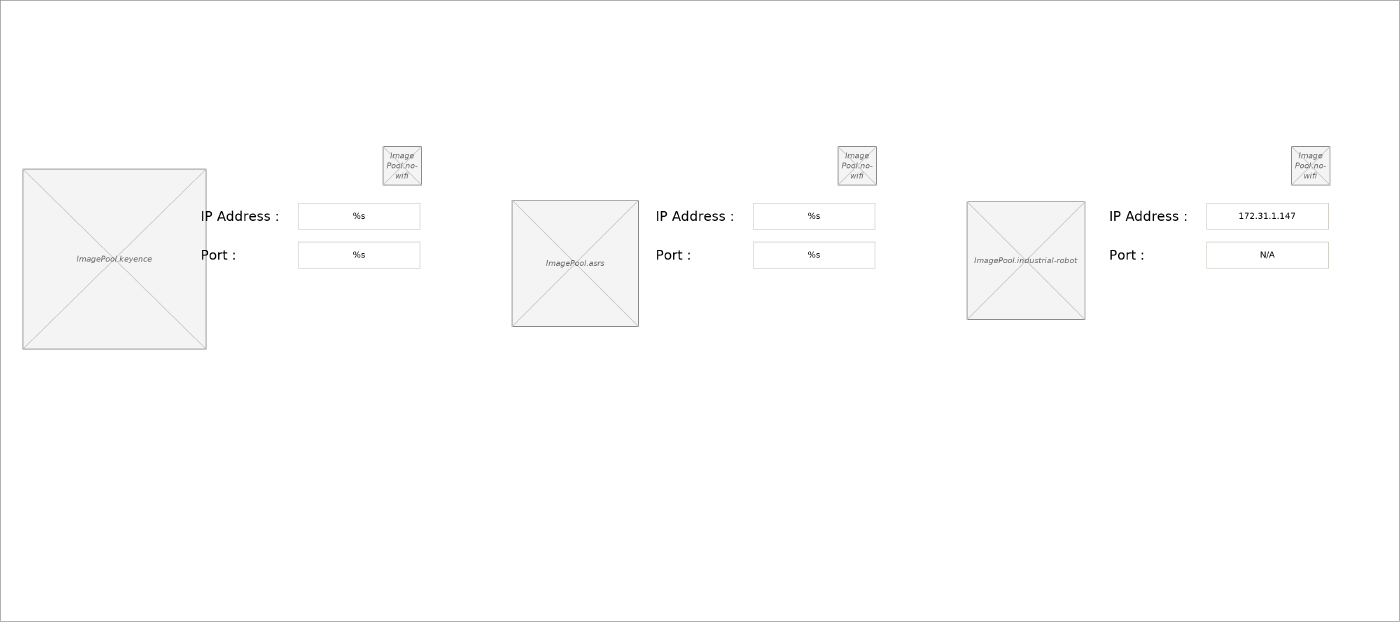
VISUALIZATION NETWORK_CONTENT  // 1800x800
    Rectangle (0,0 1800x800)
    Group (29,83 545x416)
        RoundedRectangle (5,86 540x330)
        Image (0,134 236x232), image: ImagePool.keyence
        Image (463,105 50x50), invisible if: not IO.fbClient_QR.bConnected, image: ImagePool.wifi
        Label (69,0 420x66), "KEYENCE Scanner"
        Label (226,178 126x34), "IP Address :"
        Textfield (354,178 157x34), "%s", text variable: IO.fbClient_QR.sRemoteHost
        Label (226,228 126x34), "Port :"
        Textfield (354,228 157x34), "%s", text variable: IO.fbClient_QR.nRemotePort
        Image (463,105 50x50), invisible if: IO.fbClient_QR.bConnected, image: ImagePool.no-wifi
    Group (619,83 540x436)
        RoundedRectangle (0,86 540x350)
        Image (458,105 50x50), invisible if: not IO.fbClient_ASRS.bConnected, image: ImagePool.wifi
        Label (64,0 420x66), "WCS Server"
        Label (221,178 126x34), "IP Address :"
        Textfield (349,178 157x34), "%s", text variable: IO.fbClient_ASRS.sRemoteHost
        Label (221,228 126x34), "Port :"
        Textfield (349,228 157x34), "%s", text variable: IO.fbClient_ASRS.nRemotePort
        Image (39,174 163x163), image: ImagePool.asrs
        Image (458,105 50x50), invisible if: IO.fbClient_ASRS.bConnected, image: ImagePool.no-wifi
    Group (1202,83 540x436)
        RoundedRectangle (0,86 540x350)
        Image (458,105 50x50), invisible if: not IO_KUKA.bPro_act, image: ImagePool.wifi
        Label (64,0 420x66), "KUKA Robot"
        Label (221,178 126x34), "IP Address :"
        Textfield (349,178 157x34), "172.31.1.147"
        Label (221,228 126x34), "Port :"
        Textfield (349,228 157x34), "N/A"
        Image (41,176 152x152), image: ImagePool.industrial-robot
        Image (458,105 50x50), invisible if: IO_KUKA.bPro_act, image: ImagePool.no-wifi
END_VISUALIZATION

(* stored: Version 1.1.0.1, ProductVersion 3.1.4024.12
   Visu NETWORK_CONTENT: Id {24ac47b5-de0c-4655-91da-44e3088b9c09} *)
